# EPICS substitutions: iocs/piJenaIOC/iocBoot/iocPiJena/PiJenaAsyn.substitutions
# file "$(MOTOR)/db/motor.db"
# {
# pattern
# {P,       N,	 M,	    DTYP,         C,      S,	DESC,		EGU,	DIR,    VELO,VBAS,  ACCL,	   BDST,	 BVEL,	BACC,	MRES,	PREC,	DHLM,	DLLM, INIT}
# {piJena:, 1,     "m$(N)",  "PIJEDS",      0,      0,    "motor $(N)",   um,     Pos,    2.,   0,     .2,             0,           0,    .2,      .001,   5,      100,    0,   ""}
# {piJena:, 2,     "m$(N)",  "PIJEDS",      0,      1,    "motor $(N)",   um,     Pos,    2.,   0,     .2,             0,           0,    .2,      .001,   5,      100,    0,   ""}
# }

file "$(MOTOR)/db/asyn_motor.db"
{
pattern
{N,   M,       DTYP,         PORT,    ADDR,  DESC,          EGU,  DIR,  VELO,  VBAS,  ACCL,  BDST,  BVEL,  BACC,  MRES,  PREC, DHLM,  DLLM, RTRY, INIT}
{1,  "m$(N)",  "asynMotor",  JENA1,      0,  "motor $(N)",  um,   Pos,     1,   .1,     .2,     0,     1,    .2,  0.001,   6,  100,  -100,    0,   ""}
{2,  "m$(N)",  "asynMotor",  JENA1,      1,  "motor $(N)",  um,   Pos,     1,   .1,     .2,     0,     1,    .2,  0.001,   6,  100,  -100,    0,   ""}
{3,  "m$(N)",  "asynMotor",  JENA1,      2,  "motor $(N)",  um,   Pos,     1,   .1,     .2,     0,     1,    .2,  0.001,   6,  100,  -100,    0,   ""}
}
